// TIA Portal project "AWL LIBRO 6" (V11)

(* hardware
DEVICE "S7300/ET200 station_1"  SIMATIC 300-Station
   slot 0: "Perfil soporte_0"  Rail  6ES7 390-1***0-0AA0
   slot 2: "PLC_1"  CPU 313C-2 DP  6ES7 313-6CF03-0AB0  V2.6
      slot 0: "Interfaz MPI_1"  MPI
      slot 1: "Interfaz DP_1"  DP
      slot 2: "DI16/DO16_1"  DI16/DO16
      slot 4: "Contaje_1"  Counter
*)

// ===== PLC "PLC_1"  CPU 313C-2 DP =====

VAR_GLOBAL   // PLC tag table "Tabla de variables estándar"
   "1" AT %E0.0 : Bool;
   "2" AT %E0.1 : Bool;
   "3" AT %E0.2 : Bool;
   "4" AT %E0.3 : Bool;
   "5" AT %E0.4 : Bool;
   "6" AT %E0.5 : Bool;
   "7" AT %E0.6 : Bool;
   "8" AT %E0.7 : Bool;
   "9" AT %E1.0 : Bool;
   "0" AT %E1.1 : Bool;
   "ON" AT %E1.2 : Bool;
   "OFF" AT %E1.3 : Bool;
   "CONTADOR" AT %MW10 : Int;
   "CONTACTO MAGNETICO" AT %A0.0 : Bool;
   "T0" AT %T0 : Timer;
   "INTERMITENCIA" AT %M100.5 : Bool;
   "ALARMA" AT %A0.1 : Bool;
   "T1" AT %T1 : Timer;
   "T2" AT %T2 : Timer;
END_VAR

DATA_BLOCK "F Y B"   // DB1
{ S7_Optimized_Access := 'FALSE' }
VERSION : 0.1
   VAR
      F0 : Bool;
      F1 : Bool;
      F2 : Bool;
      F3 : Bool;
      F4 : Bool;
      F5 : Bool;
      F6 : Bool;
      F7 : Bool;
      F8 : Bool;
      F9 : Bool;
      F10 : Bool;
      B0 : Bool;
      B1 : Bool;
      B2 : Bool;
      B3 : Bool;
      B4 : Bool;
      B5 : Bool;
      B6 : Bool;
      B7 : Bool;
      B8 : Bool;
      B9 : Bool;
      B10 : Bool;
      "CONTADOR U.MILLAR." : Int;
      "R UM" : Int;
      "CONTADOR CENTENAS." : Int;
      "R C" : Int;
      "CONTADOR DECENAS." : Int;
      "R D" : Int;
      "CONTADOR UNIDADES." : Int;
      "R U" : Int;
   END_VAR
BEGIN
END_DATA_BLOCK

ORGANIZATION_BLOCK "Main"   // OB1, STL
TITLE = EJERCICIO 6. / "Main Program Sweep (Cycle)"
{ S7_Optimized_Access := 'FALSE' }
VERSION : 0.1
   VAR_TEMP
      OB1_EV_CLASS : Byte;   // Bits 0-3 = 1 (Coming event), Bits 4-7 = 1 (Event class 1)
      OB1_SCAN_1 : Byte;   // 1 (Cold restart scan 1 of OB 1), 3 (Scan 2-n of OB 1)
      OB1_PRIORITY : Byte;   // Priority of OB Execution
      OB1_OB_NUMBR : Byte;   // 1 (Organization block 1, OB1)
      OB1_RESERVED_1 : Byte;   // Reserved for system
      OB1_RESERVED_2 : Byte;   // Reserved for system
      OB1_PREV_CYCLE : Int;   // Cycle time of previous OB1 scan (milliseconds)
      OB1_MIN_CYCLE : Int;   // Minimum cycle time of OB1 (milliseconds)
      OB1_MAX_CYCLE : Int;   // Maximum cycle time of OB1 (milliseconds)
      OB1_DATE_TIME : Date_And_Time;   // Date and time OB1 started
   END_VAR
BEGIN
END_ORGANIZATION_BLOCK